// TIA Portal V16 export
// export: Created 2023-10-30T22:43:47.694868Z, ExportSetting WithDefaults, DisplayName Totally Integrated Automation Portal, DisplayVersion V16, DisplayName TIA Portal Version Control Interface, DisplayVersion V16, DisplayName TIA Portal Openness, DisplayVersion V16, DisplayName SINAMICS Startdrive Advanced, DisplayVersion V16, DisplayName SINAMICS Startdrive G130, G150, S120, S150, SINAMICS MV, S210, DisplayVersion V16, DisplayName SINAMICS Startdrive G110M, G120, G120C, G120D, G120P, DisplayVersion V16, DisplayName STEP 7 Professional, DisplayVersion V16, DisplayName STEP 7 Safety, DisplayVersion V16, DisplayName WinCC Professional, DisplayVersion V16
ORGANIZATION_BLOCK "Main"   // OB1, LAD, ProgramCycle
TITLE = "Main Program Sweep (Cycle)"
{ S7_Optimized_Access := 'TRUE' }
VERSION : 0.1
// stored: AutoNumber true, IsIECCheckEnabled false, SetENOAutomatically false
   VAR_INPUT
      Initial_Call : Bool;   // Initial call of this OB
      Remanence : Bool;   // =True, if remanent data are available
   END_VAR
   VAR_TEMP   // added for the SCL form of the ladder/FBD networks
      _w1 : Bool;
      _w2 : Bool;
      _w3 : Bool;
      _w4 : Bool;
   END_VAR
BEGIN

REGION Network 1: Control Maestro
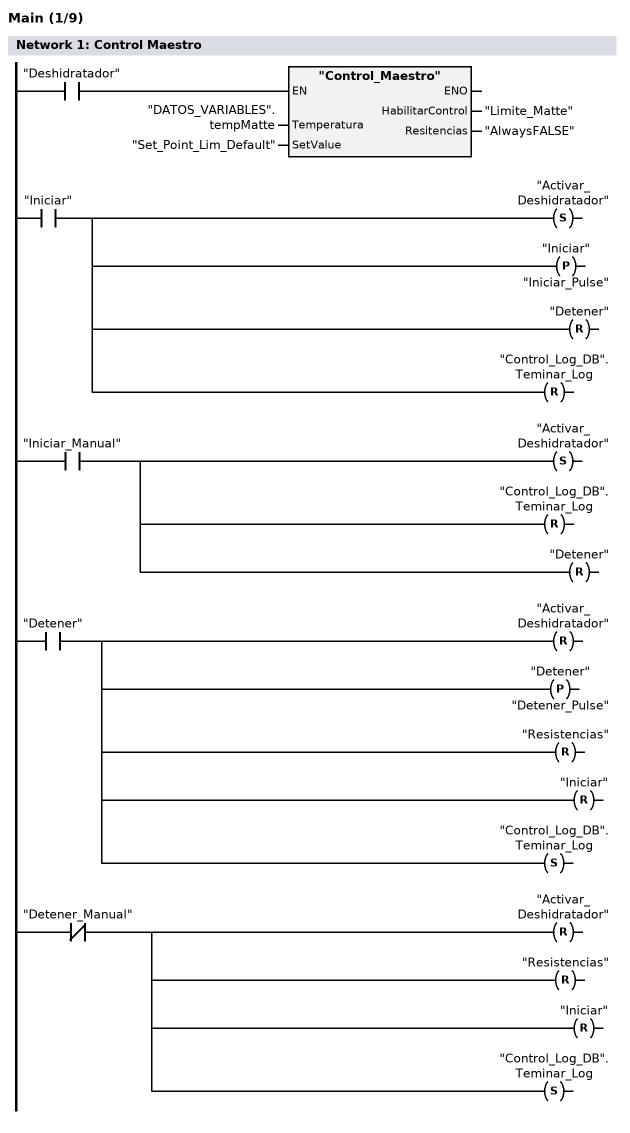
   IF "Deshidratador" THEN
       "Control_Maestro"(Temperatura := "DATOS_VARIABLES".tempMatte,
                         SetValue := "Set_Point_Lim_Default",
                         HabilitarControl => "Limite_Matte",
                         Resitencias => "AlwaysFALSE");
   END_IF;
   IF "Iniciar" THEN "Activar_Deshidratador" := TRUE; END_IF;
   #_w1 := "Iniciar";
   #_w2 := "Iniciar";
   "Iniciar" := #_w1 AND NOT "Iniciar_Pulse";   // rising edge
   "Iniciar_Pulse" := #_w1;
   IF #_w2 THEN
       "Detener" := FALSE;
       "Control_Log_DB".Teminar_Log := FALSE;
   END_IF;
   IF "Iniciar_Manual" THEN
       "Activar_Deshidratador" := TRUE;
       "Control_Log_DB".Teminar_Log := FALSE;
       "Detener" := FALSE;
   END_IF;
   IF "Detener" THEN "Activar_Deshidratador" := FALSE; END_IF;
   #_w3 := "Detener";
   #_w4 := "Detener";
   "Detener" := #_w3 AND NOT "Detener_Pulse";   // rising edge
   "Detener_Pulse" := #_w3;
   IF #_w4 THEN
       "Resistencias" := FALSE;
       "Iniciar" := FALSE;
       "Control_Log_DB".Teminar_Log := TRUE;
   END_IF;
   IF NOT "Detener_Manual" THEN
       "Activar_Deshidratador" := FALSE;
       "Resistencias" := FALSE;
       "Iniciar" := FALSE;
       "Control_Log_DB".Teminar_Log := TRUE;
   END_IF;
END_REGION

REGION Network 2: Matte
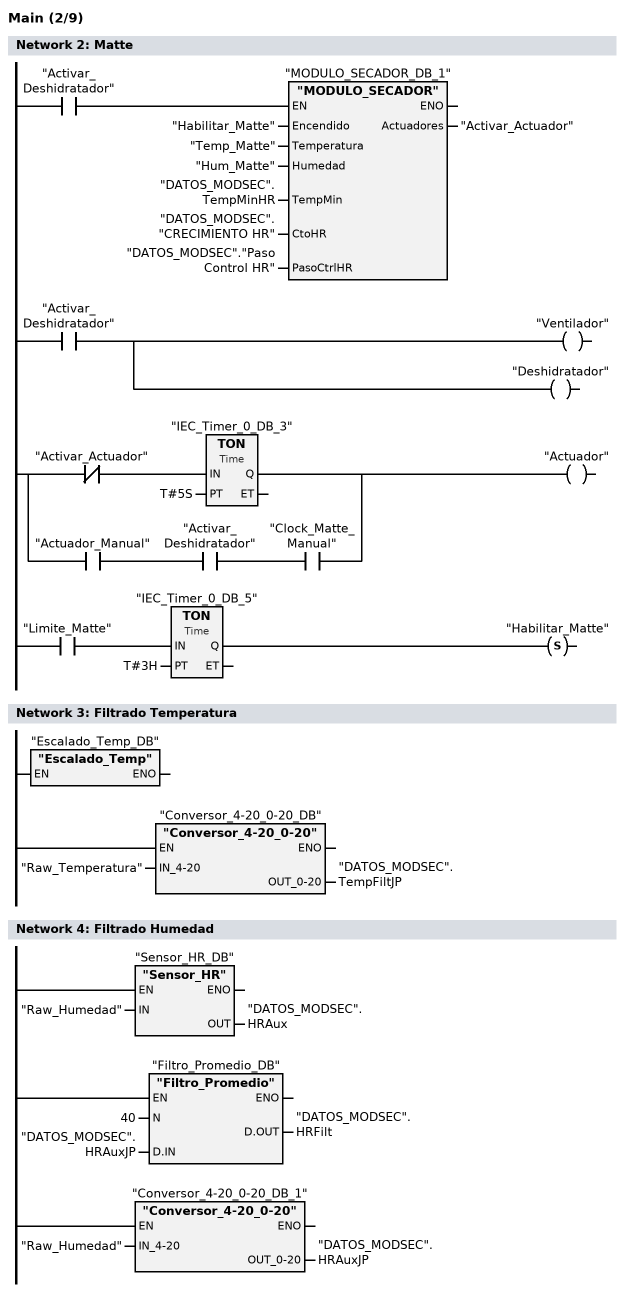
   RUNG wire#powerrail
      Contact( "Activar_Deshidratador" )
      "MODULO_SECADOR_DB_1"(Encendido := "Habilitar_Matte", Temperatura := "Temp_Matte", Humedad := "Hum_Matte", TempMin := "DATOS_MODSEC".TempMinHR, CtoHR := "DATOS_MODSEC"."CRECIMIENTO HR", PasoCtrlHR := "DATOS_MODSEC"."Paso Control HR", Actuadores => "Activar_Actuador")
   END_RUNG
   RUNG wire#powerrail
      Contact( "Activar_Deshidratador" )
      wire#w1
      Coil( "Ventilador" )
   END_RUNG
   RUNG wire#w1
      Coil( "Deshidratador" )
   END_RUNG
   RUNG wire#powerrail
      I_Contact( "Activar_Actuador" )
      { S7_Templates := "time_type := Time" } "IEC_Timer_0_DB_3".TON(pt := T#5S, et =>)
      wire#w2
      Coil( "Actuador" )
   END_RUNG
   RUNG wire#powerrail
      Contact( "Actuador_Manual" )
      Contact( "Activar_Deshidratador" )
      Contact( "Clock_Matte_Manual" )
   END_RUNG wire#w2
   RUNG wire#powerrail
      Contact( "Limite_Matte" )
      { S7_Templates := "time_type := Time" } "IEC_Timer_0_DB_5".TON(pt := T#3H, et =>)
      S_Coil( "Habilitar_Matte" )
   END_RUNG
   // the same network as SCL:
   IF "Activar_Deshidratador" THEN
       "MODULO_SECADOR_DB_1"(Encendido := "Habilitar_Matte",   // "MODULO_SECADOR"
                             Temperatura := "Temp_Matte",
                             Humedad := "Hum_Matte",
                             TempMin := "DATOS_MODSEC".TempMinHR,
                             CtoHR := "DATOS_MODSEC"."CRECIMIENTO HR",
                             PasoCtrlHR := "DATOS_MODSEC"."Paso Control HR",
                             Actuadores => "Activar_Actuador");
   END_IF;
   "Ventilador" := "Activar_Deshidratador";
   "Deshidratador" := "Activar_Deshidratador";
   "IEC_Timer_0_DB_3".TON(IN := NOT "Activar_Actuador", PT := T#5S);
   "Actuador" := "IEC_Timer_0_DB_3".Q OR ("Actuador_Manual" AND "Activar_Deshidratador" AND "Clock_Matte_Manual");
   "IEC_Timer_0_DB_5".TON(IN := "Limite_Matte", PT := T#3H);
   IF "IEC_Timer_0_DB_5".Q THEN "Habilitar_Matte" := TRUE; END_IF;
END_REGION

REGION Network 3: Filtrado Temperatura
   RUNG wire#powerrail
      "Escalado_Temp_DB"()
   END_RUNG
   RUNG wire#powerrail
      "Conversor_4-20_0-20_DB"("IN_4-20" := "Raw_Temperatura", "OUT_0-20" => "DATOS_MODSEC".TempFiltJP)
   END_RUNG
   // the same network as SCL:
   "Escalado_Temp_DB"();   // "Escalado_Temp"
   "Conversor_4-20_0-20_DB"("IN_4-20" := "Raw_Temperatura", "OUT_0-20" => "DATOS_MODSEC".TempFiltJP);   // "Conversor_4-20_0-20"
END_REGION

REGION Network 4: Filtrado Humedad
   RUNG wire#powerrail
      "Sensor_HR_DB"(IN := "Raw_Humedad", OUT => "DATOS_MODSEC".HRAux)
   END_RUNG
   RUNG wire#powerrail
      "Filtro_Promedio_DB"(N := 40, "D.IN" := "DATOS_MODSEC".HRAuxJP, "D.OUT" => "DATOS_MODSEC".HRFilt)
   END_RUNG
   RUNG wire#powerrail
      "Conversor_4-20_0-20_DB_1"("IN_4-20" := "Raw_Humedad", "OUT_0-20" => "DATOS_MODSEC".HRAuxJP)
   END_RUNG
   // the same network as SCL:
   "Sensor_HR_DB"(IN := "Raw_Humedad", OUT => "DATOS_MODSEC".HRAux);   // "Sensor_HR"
   "Filtro_Promedio_DB"(N := 40, "D.IN" := "DATOS_MODSEC".HRAuxJP, "D.OUT" => "DATOS_MODSEC".HRFilt);   // "Filtro_Promedio"
   "Conversor_4-20_0-20_DB_1"("IN_4-20" := "Raw_Humedad", "OUT_0-20" => "DATOS_MODSEC".HRAuxJP);   // "Conversor_4-20_0-20"
END_REGION

REGION Network 5: Simulación
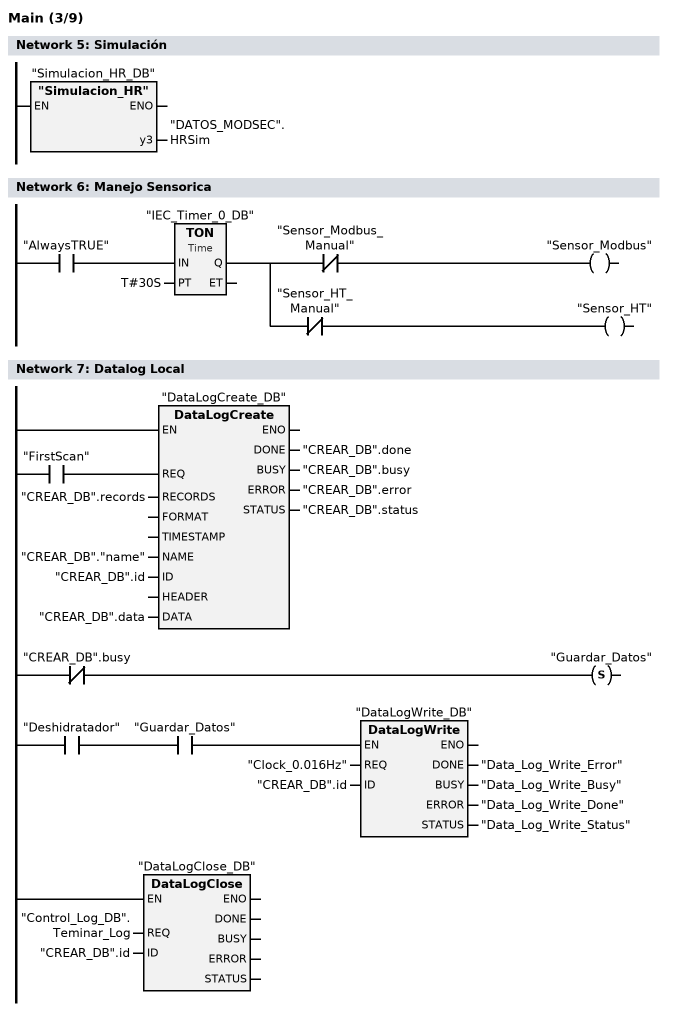
   RUNG wire#powerrail
      "Simulacion_HR_DB"(y3 => "DATOS_MODSEC".HRSim)
   END_RUNG
   // the same network as SCL:
   "Simulacion_HR_DB"(y3 => "DATOS_MODSEC".HRSim);   // "Simulacion_HR"
END_REGION

REGION Network 6: Manejo Sensorica
   RUNG wire#powerrail
      Contact( "AlwaysTRUE" )
      { S7_Templates := "time_type := Time" } "IEC_Timer_0_DB".TON(pt := T#30S, et =>)
      wire#w1
      I_Contact( "Sensor_Modbus_Manual" )
      Coil( "Sensor_Modbus" )
   END_RUNG
   RUNG wire#w1
      I_Contact( "Sensor_HT_Manual" )
      Coil( "Sensor_HT" )
   END_RUNG
   // the same network as SCL:
   "IEC_Timer_0_DB".TON(IN := "AlwaysTRUE", PT := T#30S);
   "Sensor_Modbus" := "IEC_Timer_0_DB".Q AND NOT "Sensor_Modbus_Manual";
   "Sensor_HT" := "IEC_Timer_0_DB".Q AND NOT "Sensor_HT_Manual";
END_REGION

REGION Network 7: Datalog Local
   RUNG wire#powerrail
      "DataLogCreate_DB".DataLogCreate(REQ := wire#w1, RECORDS := "CREAR_DB".records, FORMAT :=, TIMESTAMP :=, "NAME" := "CREAR_DB"."name", ID := "CREAR_DB".id, HEADER :=, DATA := "CREAR_DB".data, DONE => "CREAR_DB".done, BUSY => "CREAR_DB".busy, ERROR => "CREAR_DB".error, STATUS => "CREAR_DB".status)
   END_RUNG
   RUNG wire#powerrail
      Contact( "FirstScan" )
   END_RUNG wire#w1
   RUNG wire#powerrail
      I_Contact( "CREAR_DB".busy )
      S_Coil( "Guardar_Datos" )
   END_RUNG
   RUNG wire#powerrail
      Contact( "Deshidratador" )
      Contact( "Guardar_Datos" )
      "DataLogWrite_DB".DataLogWrite(REQ := "Clock_0.016Hz", ID := "CREAR_DB".id, DONE => "Data_Log_Write_Error", BUSY => "Data_Log_Write_Busy", ERROR => "Data_Log_Write_Done", STATUS => "Data_Log_Write_Status")
   END_RUNG
   RUNG wire#powerrail
      "DataLogClose_DB".DataLogClose(REQ := "Control_Log_DB".Teminar_Log, ID := "CREAR_DB".id, DONE =>, BUSY =>, ERROR =>, STATUS =>)
   END_RUNG
   // the same network as SCL:
   "DataLogCreate_DB"(REQ := "FirstScan",   // DataLogCreate
                      RECORDS := "CREAR_DB".records,
                      "NAME" := "CREAR_DB"."name",
                      ID := "CREAR_DB".id,
                      DATA := "CREAR_DB".data,
                      DONE => "CREAR_DB".done,
                      BUSY => "CREAR_DB".busy,
                      ERROR => "CREAR_DB".error,
                      STATUS => "CREAR_DB".status);
   IF NOT "CREAR_DB".busy THEN "Guardar_Datos" := TRUE; END_IF;
   IF "Deshidratador" AND "Guardar_Datos" THEN
       "DataLogWrite_DB"(REQ := "Clock_0.016Hz",   // DataLogWrite
                         ID := "CREAR_DB".id,
                         DONE => "Data_Log_Write_Error",
                         BUSY => "Data_Log_Write_Busy",
                         ERROR => "Data_Log_Write_Done",
                         STATUS => "Data_Log_Write_Status");
   END_IF;
   "DataLogClose_DB"(REQ := "Control_Log_DB".Teminar_Log, ID := "CREAR_DB".id);   // DataLogClose
END_REGION

REGION Network 8: Mover Datos para Log Remoto
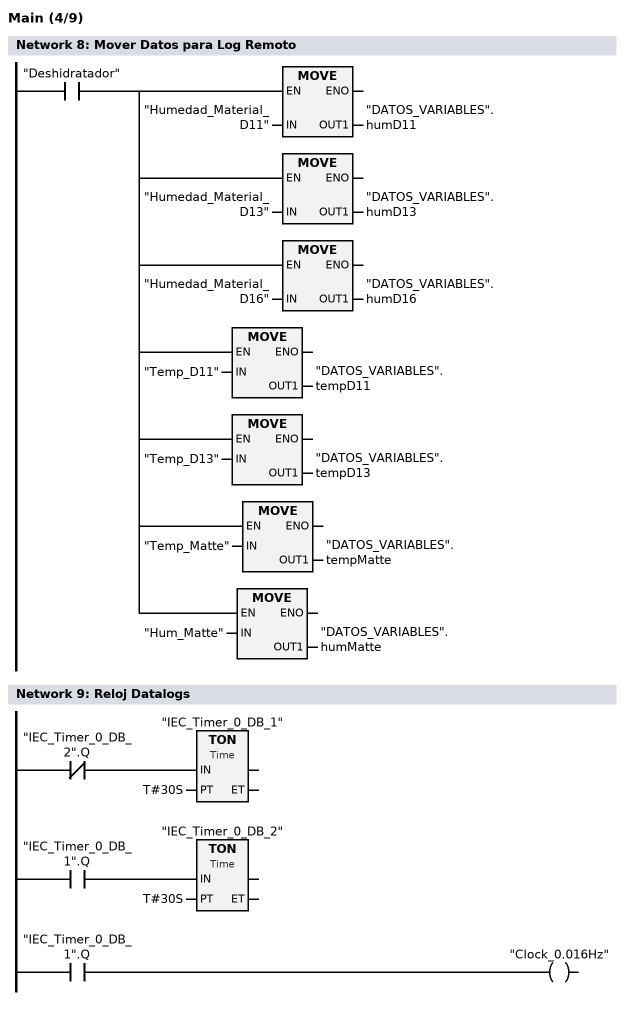
   RUNG wire#powerrail
      Contact( "Deshidratador" )
      wire#w1
      Move(in := "Humedad_Material_D11", out1 => "DATOS_VARIABLES".humD11)
   END_RUNG
   RUNG wire#w1
      Move(in := "Humedad_Material_D13", out1 => "DATOS_VARIABLES".humD13)
   END_RUNG
   RUNG wire#w1
      Move(in := "Humedad_Material_D16", out1 => "DATOS_VARIABLES".humD16)
   END_RUNG
   RUNG wire#w1
      Move(in := "Temp_D11", out1 => "DATOS_VARIABLES".tempD11)
   END_RUNG
   RUNG wire#w1
      Move(in := "Temp_D13", out1 => "DATOS_VARIABLES".tempD13)
   END_RUNG
   RUNG wire#w1
      Move(in := "Temp_Matte", out1 => "DATOS_VARIABLES".tempMatte)
   END_RUNG
   RUNG wire#w1
      Move(in := "Hum_Matte", out1 => "DATOS_VARIABLES".humMatte)
   END_RUNG
   // the same network as SCL:
   IF "Deshidratador" THEN
       "DATOS_VARIABLES".humD11 := "Humedad_Material_D11";
       "DATOS_VARIABLES".humD13 := "Humedad_Material_D13";
       "DATOS_VARIABLES".humD16 := "Humedad_Material_D16";
       "DATOS_VARIABLES".tempD11 := "Temp_D11";
       "DATOS_VARIABLES".tempD13 := "Temp_D13";
       "DATOS_VARIABLES".tempMatte := "Temp_Matte";
       "DATOS_VARIABLES".humMatte := "Hum_Matte";
   END_IF;
END_REGION

REGION Network 9: Reloj Datalogs
   RUNG wire#powerrail
      I_Contact( "IEC_Timer_0_DB_2".Q )
      { S7_Templates := "time_type := Time" } "IEC_Timer_0_DB_1".TON(pt := T#30S, et =>)
   END_RUNG
   RUNG wire#powerrail
      Contact( "IEC_Timer_0_DB_1".Q )
      { S7_Templates := "time_type := Time" } "IEC_Timer_0_DB_2".TON(pt := T#30S, et =>)
   END_RUNG
   RUNG wire#powerrail
      Contact( "IEC_Timer_0_DB_1".Q )
      Coil( "Clock_0.016Hz" )
   END_RUNG
   // the same network as SCL:
   "IEC_Timer_0_DB_1".TON(IN := NOT "IEC_Timer_0_DB_2".Q, PT := T#30S);
   "IEC_Timer_0_DB_2".TON(IN := "IEC_Timer_0_DB_1".Q, PT := T#30S);
   "Clock_0.016Hz" := "IEC_Timer_0_DB_1".Q;
END_REGION

REGION Network 10: Mover Datos para Log Local
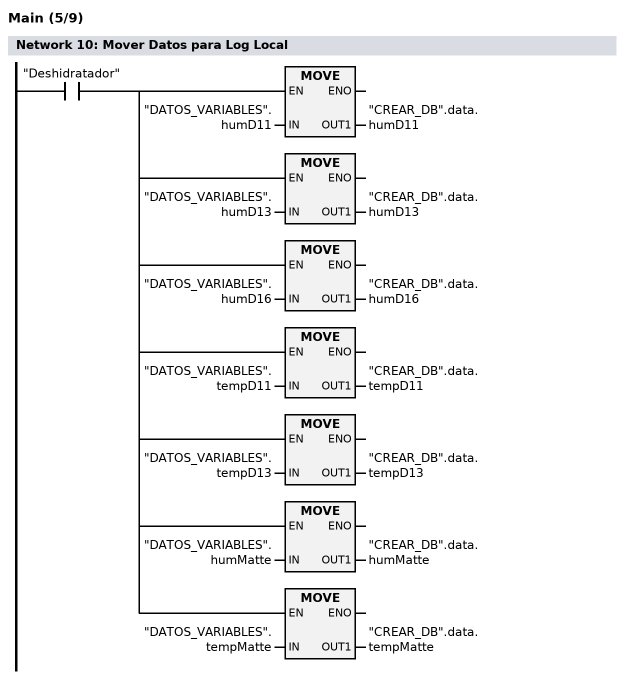
   RUNG wire#powerrail
      Contact( "Deshidratador" )
      wire#w1
      Move(in := "DATOS_VARIABLES".humD11, out1 => "CREAR_DB".data.humD11)
   END_RUNG
   RUNG wire#w1
      Move(in := "DATOS_VARIABLES".humD13, out1 => "CREAR_DB".data.humD13)
   END_RUNG
   RUNG wire#w1
      Move(in := "DATOS_VARIABLES".humD16, out1 => "CREAR_DB".data.humD16)
   END_RUNG
   RUNG wire#w1
      Move(in := "DATOS_VARIABLES".tempD11, out1 => "CREAR_DB".data.tempD11)
   END_RUNG
   RUNG wire#w1
      Move(in := "DATOS_VARIABLES".tempD13, out1 => "CREAR_DB".data.tempD13)
   END_RUNG
   RUNG wire#w1
      Move(in := "DATOS_VARIABLES".humMatte, out1 => "CREAR_DB".data.humMatte)
   END_RUNG
   RUNG wire#w1
      Move(in := "DATOS_VARIABLES".tempMatte, out1 => "CREAR_DB".data.tempMatte)
   END_RUNG
   // the same network as SCL:
   IF "Deshidratador" THEN
       "CREAR_DB".data.humD11 := "DATOS_VARIABLES".humD11;
       "CREAR_DB".data.humD13 := "DATOS_VARIABLES".humD13;
       "CREAR_DB".data.humD16 := "DATOS_VARIABLES".humD16;
       "CREAR_DB".data.tempD11 := "DATOS_VARIABLES".tempD11;
       "CREAR_DB".data.tempD13 := "DATOS_VARIABLES".tempD13;
       "CREAR_DB".data.humMatte := "DATOS_VARIABLES".humMatte;
       "CREAR_DB".data.tempMatte := "DATOS_VARIABLES".tempMatte;
   END_IF;
END_REGION

REGION Network 11: Comunicación Modbus
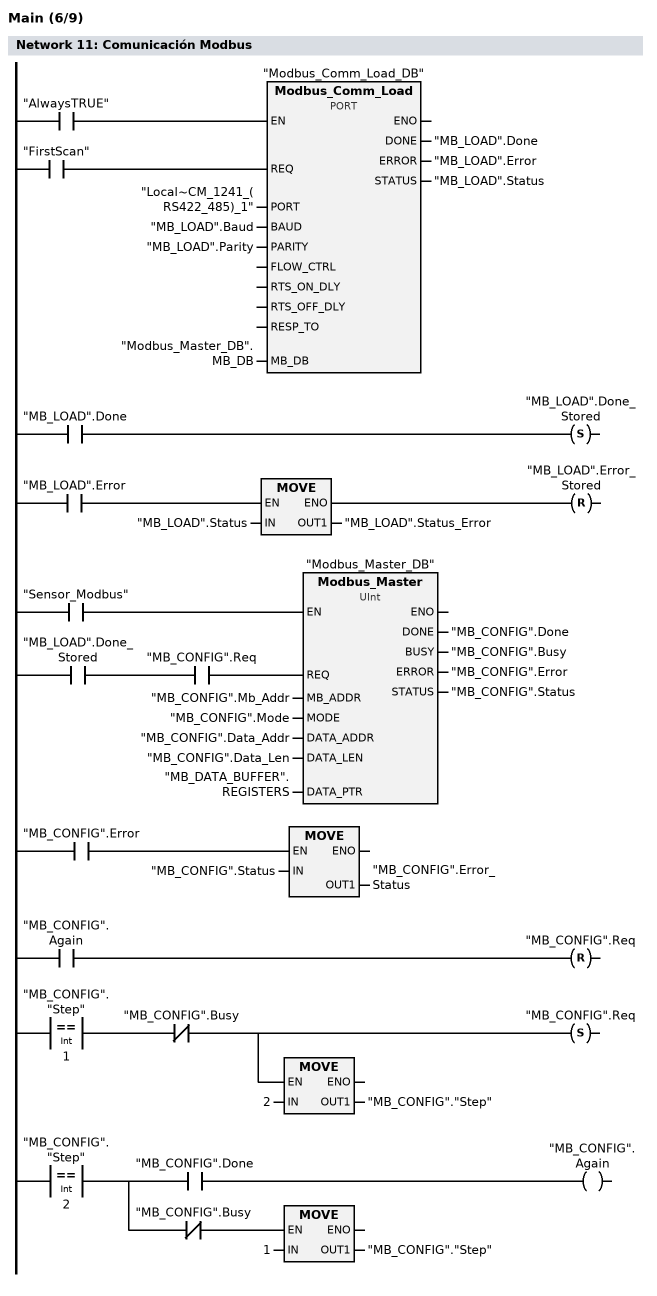
   RUNG wire#powerrail
      Contact( "AlwaysTRUE" )
      { S7_Templates := "[card := 0, port_type := PORT, word_type := UInt, dint_type := UDInt, mbbase_type := P2P_MB_BASE]" } "Modbus_Comm_Load_DB".Modbus_Comm_Load(REQ := wire#w1, PORT := "Local~CM_1241_(RS422_485)_1", BAUD := "MB_LOAD".Baud, PARITY := "MB_LOAD".Parity, FLOW_CTRL :=, RTS_ON_DLY :=, RTS_OFF_DLY :=, RESP_TO :=, MB_DB := "Modbus_Master_DB".MB_DB, DONE => "MB_LOAD".Done, ERROR => "MB_LOAD".Error, STATUS => "MB_LOAD".Status)
   END_RUNG
   RUNG wire#powerrail
      Contact( "FirstScan" )
   END_RUNG wire#w1
   RUNG wire#powerrail
      Contact( "MB_LOAD".Done )
      S_Coil( "MB_LOAD".Done_Stored )
   END_RUNG
   RUNG wire#powerrail
      Contact( "MB_LOAD".Error )
      Move(in := "MB_LOAD".Status, out1 => "MB_LOAD".Status_Error)
      R_Coil( "MB_LOAD".Error_Stored )
   END_RUNG
   RUNG wire#powerrail
      Contact( "Sensor_Modbus" )
      { S7_Templates := "[card := 0, word_type := UInt, dword_type := UDInt, byte_type := USInt, any_type := Variant]" } "Modbus_Master_DB".Modbus_Master(REQ := wire#w2, MB_ADDR := "MB_CONFIG".Mb_Addr, MODE := "MB_CONFIG".Mode, DATA_ADDR := "MB_CONFIG".Data_Addr, DATA_LEN := "MB_CONFIG".Data_Len, DATA_PTR := "MB_DATA_BUFFER".REGISTERS, DONE => "MB_CONFIG".Done, BUSY => "MB_CONFIG".Busy, ERROR => "MB_CONFIG".Error, STATUS => "MB_CONFIG".Status)
   END_RUNG
   RUNG wire#powerrail
      Contact( "MB_LOAD".Done_Stored )
      Contact( "MB_CONFIG".Req )
   END_RUNG wire#w2
   RUNG wire#powerrail
      Contact( "MB_CONFIG".Error )
      Move(in := "MB_CONFIG".Status, out1 => "MB_CONFIG".Error_Status)
   END_RUNG
   RUNG wire#powerrail
      Contact( "MB_CONFIG".Again )
      R_Coil( "MB_CONFIG".Req )
   END_RUNG
   RUNG wire#powerrail
      { S7_Templates := "SrcType := Int" } EQ_Contact(in1 := "MB_CONFIG"."Step", in2 := 1)
      I_Contact( "MB_CONFIG".Busy )
      wire#w3
      S_Coil( "MB_CONFIG".Req )
   END_RUNG
   RUNG wire#w3
      Move(in := 2, out1 => "MB_CONFIG"."Step")
   END_RUNG
   RUNG wire#powerrail
      { S7_Templates := "SrcType := Int" } EQ_Contact(in1 := "MB_CONFIG"."Step", in2 := 2)
      wire#w4
      Contact( "MB_CONFIG".Done )
      Coil( "MB_CONFIG".Again )
   END_RUNG
   RUNG wire#w4
      I_Contact( "MB_CONFIG".Busy )
      Move(in := 1, out1 => "MB_CONFIG"."Step")
   END_RUNG
   // the same network as SCL:
   IF "AlwaysTRUE" THEN
       "Modbus_Comm_Load_DB"(REQ := "FirstScan",   // Modbus_Comm_Load
                             PORT := "Local~CM_1241_(RS422_485)_1",
                             BAUD := "MB_LOAD".Baud,
                             PARITY := "MB_LOAD".Parity,
                             MB_DB := "Modbus_Master_DB".MB_DB,
                             DONE => "MB_LOAD".Done,
                             ERROR => "MB_LOAD".Error,
                             STATUS => "MB_LOAD".Status);
   END_IF;
   IF "MB_LOAD".Done THEN "MB_LOAD".Done_Stored := TRUE; END_IF;
   IF "MB_LOAD".Error THEN
       "MB_LOAD".Status_Error := "MB_LOAD".Status;
       "MB_LOAD".Error_Stored := FALSE;
   END_IF;
   IF "Sensor_Modbus" THEN
       "Modbus_Master_DB"(REQ := "MB_LOAD".Done_Stored AND "MB_CONFIG".Req,   // Modbus_Master
                          MB_ADDR := "MB_CONFIG".Mb_Addr,
                          MODE := "MB_CONFIG".Mode,
                          DATA_ADDR := "MB_CONFIG".Data_Addr,
                          DATA_LEN := "MB_CONFIG".Data_Len,
                          DATA_PTR := "MB_DATA_BUFFER".REGISTERS,
                          DONE => "MB_CONFIG".Done,
                          BUSY => "MB_CONFIG".Busy,
                          ERROR => "MB_CONFIG".Error,
                          STATUS => "MB_CONFIG".Status);
   END_IF;
   IF "MB_CONFIG".Error THEN "MB_CONFIG".Error_Status := "MB_CONFIG".Status; END_IF;
   IF "MB_CONFIG".Again THEN "MB_CONFIG".Req := FALSE; END_IF;
   IF ("MB_CONFIG"."Step" = 1) AND NOT "MB_CONFIG".Busy THEN
       "MB_CONFIG".Req := TRUE;
       "MB_CONFIG"."Step" := 2;
   END_IF;
   #_w1 := "MB_CONFIG"."Step" = 2;
   "MB_CONFIG".Again := #_w1 AND "MB_CONFIG".Done;
   IF #_w1 AND NOT "MB_CONFIG".Busy THEN "MB_CONFIG"."Step" := 1; END_IF;
END_REGION

REGION Network 12: Escalización Humedad
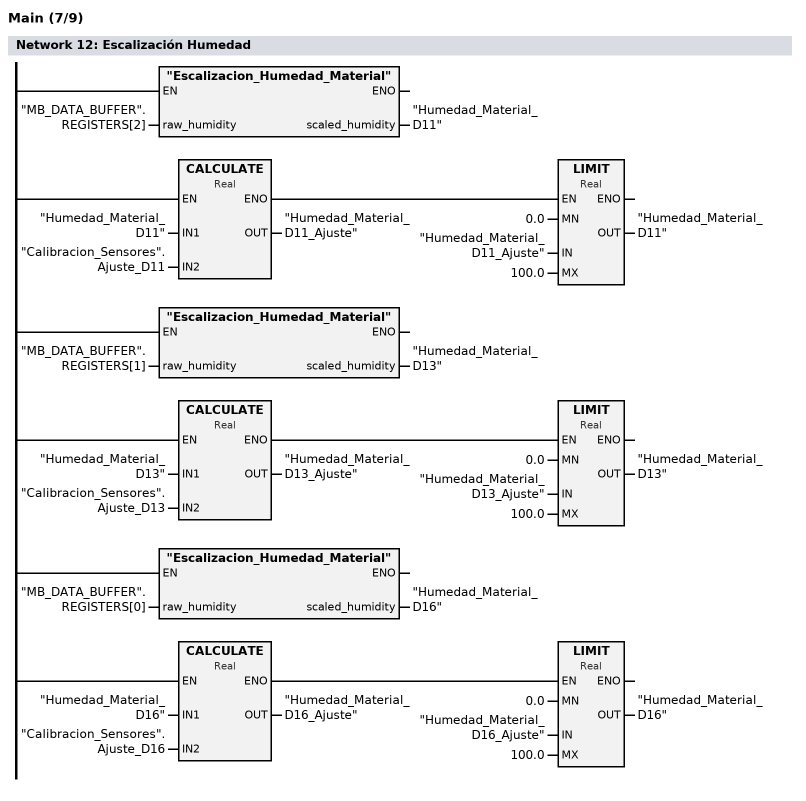
   RUNG wire#powerrail
      "Escalizacion_Humedad_Material"(raw_humidity := "MB_DATA_BUFFER".REGISTERS[2], scaled_humidity => "Humedad_Material_D11")
   END_RUNG
   RUNG wire#powerrail
      { S7_Templates := "SrcType := Real"; S7_Expression := "IN1 - IN2" } Calculate(in1 := "Humedad_Material_D11", in2 := "Calibracion_Sensores".Ajuste_D11, out => "Humedad_Material_D11_Ajuste")
      { S7_Templates := "value_type := Real" } Limit(mn := 0.0, in := "Humedad_Material_D11_Ajuste", mx := 100.0, out => "Humedad_Material_D11")
   END_RUNG
   RUNG wire#powerrail
      "Escalizacion_Humedad_Material"(raw_humidity := "MB_DATA_BUFFER".REGISTERS[1], scaled_humidity => "Humedad_Material_D13")
   END_RUNG
   RUNG wire#powerrail
      { S7_Templates := "SrcType := Real"; S7_Expression := "IN1 - IN2" } Calculate(in1 := "Humedad_Material_D13", in2 := "Calibracion_Sensores".Ajuste_D13, out => "Humedad_Material_D13_Ajuste")
      { S7_Templates := "value_type := Real" } Limit(mn := 0.0, in := "Humedad_Material_D13_Ajuste", mx := 100.0, out => "Humedad_Material_D13")
   END_RUNG
   RUNG wire#powerrail
      "Escalizacion_Humedad_Material"(raw_humidity := "MB_DATA_BUFFER".REGISTERS[0], scaled_humidity => "Humedad_Material_D16")
   END_RUNG
   RUNG wire#powerrail
      { S7_Templates := "SrcType := Real"; S7_Expression := "IN1 - IN2" } Calculate(in1 := "Humedad_Material_D16", in2 := "Calibracion_Sensores".Ajuste_D16, out => "Humedad_Material_D16_Ajuste")
      { S7_Templates := "value_type := Real" } Limit(mn := 0.0, in := "Humedad_Material_D16_Ajuste", mx := 100.0, out => "Humedad_Material_D16")
   END_RUNG
   // the same network as SCL:
   "Escalizacion_Humedad_Material"(raw_humidity := "MB_DATA_BUFFER".REGISTERS[2],
                           scaled_humidity => "Humedad_Material_D11");
   "Humedad_Material_D11_Ajuste" := "Humedad_Material_D11" - "Calibracion_Sensores".Ajuste_D11;
   "Humedad_Material_D11" := LIMIT(MN := 0.0, IN := "Humedad_Material_D11_Ajuste", MX := 100.0);
   "Escalizacion_Humedad_Material"(raw_humidity := "MB_DATA_BUFFER".REGISTERS[1],
                           scaled_humidity => "Humedad_Material_D13");
   "Humedad_Material_D13_Ajuste" := "Humedad_Material_D13" - "Calibracion_Sensores".Ajuste_D13;
   "Humedad_Material_D13" := LIMIT(MN := 0.0, IN := "Humedad_Material_D13_Ajuste", MX := 100.0);
   "Escalizacion_Humedad_Material"(raw_humidity := "MB_DATA_BUFFER".REGISTERS[0],
                           scaled_humidity => "Humedad_Material_D16");
   "Humedad_Material_D16_Ajuste" := "Humedad_Material_D16" - "Calibracion_Sensores".Ajuste_D16;
   "Humedad_Material_D16" := LIMIT(MN := 0.0, IN := "Humedad_Material_D16_Ajuste", MX := 100.0);
END_REGION

REGION Network 13: Humedad y Temperatura Deshidratador
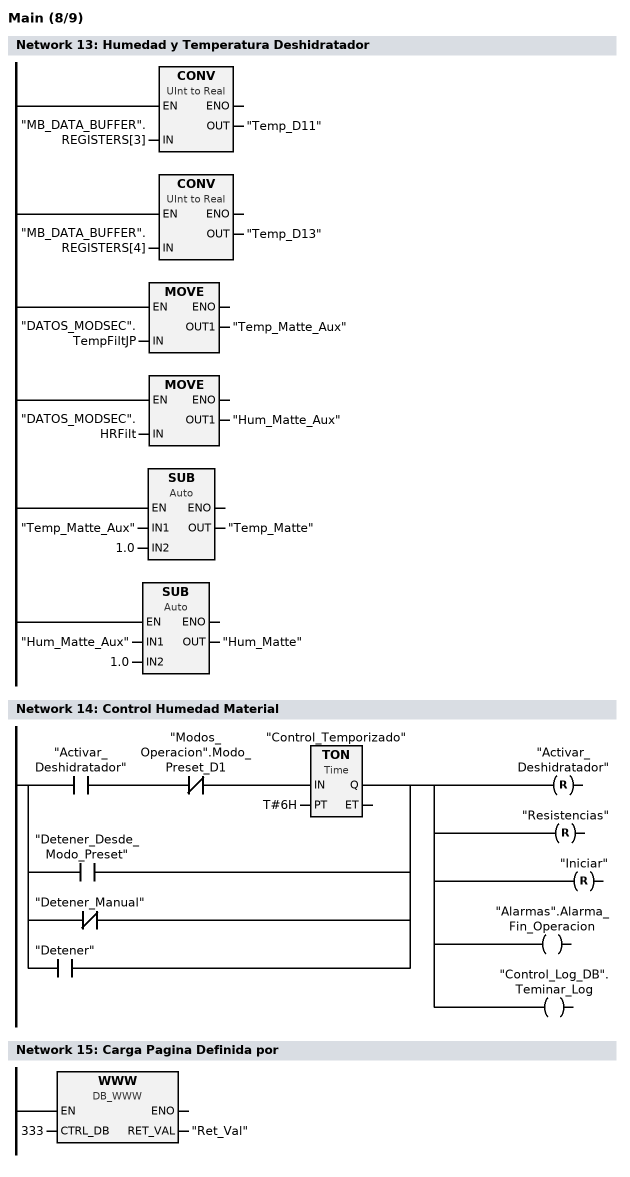
   RUNG wire#powerrail
      { S7_Templates := "[SrcType := UInt, DestType := Real]" } Convert(in := "MB_DATA_BUFFER".REGISTERS[3], out => "Temp_D11")
   END_RUNG
   RUNG wire#powerrail
      { S7_Templates := "[SrcType := UInt, DestType := Real]" } Convert(in := "MB_DATA_BUFFER".REGISTERS[4], out => "Temp_D13")
   END_RUNG
   RUNG wire#powerrail
      Move(in := "DATOS_MODSEC".TempFiltJP, out1 => "Temp_Matte_Aux")
   END_RUNG
   RUNG wire#powerrail
      Move(in := "DATOS_MODSEC".HRFilt, out1 => "Hum_Matte_Aux")
   END_RUNG
   RUNG wire#powerrail
      Sub(in1 := "Temp_Matte_Aux", in2 := 1.0, out => "Temp_Matte")
   END_RUNG
   RUNG wire#powerrail
      Sub(in1 := "Hum_Matte_Aux", in2 := 1.0, out => "Hum_Matte")
   END_RUNG
   // the same network as SCL:
   "Temp_D11" := UINT_TO_REAL("MB_DATA_BUFFER".REGISTERS[3]);
   "Temp_D13" := UINT_TO_REAL("MB_DATA_BUFFER".REGISTERS[4]);
   "Temp_Matte_Aux" := "DATOS_MODSEC".TempFiltJP;
   "Hum_Matte_Aux" := "DATOS_MODSEC".HRFilt;
   "Temp_Matte" := "Temp_Matte_Aux" - 1.0;
   "Hum_Matte" := "Hum_Matte_Aux" - 1.0;
END_REGION

REGION Network 14: Control Humedad Material
   RUNG wire#powerrail
      Contact( "Activar_Deshidratador" )
      I_Contact( "Modos_Operacion".Modo_Preset_D1 )
      { S7_Templates := "time_type := Time" } "Control_Temporizado".TON(pt := T#6H, et =>)
      wire#w1
      R_Coil( "Activar_Deshidratador" )
   END_RUNG
   RUNG wire#powerrail
      Contact( "Detener_Desde_Modo_Preset" )
   END_RUNG wire#w1
   RUNG wire#powerrail
      I_Contact( "Detener_Manual" )
   END_RUNG wire#w1
   RUNG wire#powerrail
      Contact( "Detener" )
   END_RUNG wire#w1
   RUNG wire#w1
      R_Coil( "Resistencias" )
   END_RUNG
   RUNG wire#w1
      R_Coil( "Iniciar" )
   END_RUNG
   RUNG wire#w1
      Coil( "Alarmas".Alarma_Fin_Operacion )
   END_RUNG
   RUNG wire#w1
      Coil( "Control_Log_DB".Teminar_Log )
   END_RUNG
   // the same network as SCL:
   "Control_Temporizado".TON(IN := "Activar_Deshidratador" AND NOT "Modos_Operacion".Modo_Preset_D1, PT := T#6H);
   #_w1 := "Control_Temporizado".Q OR "Detener_Desde_Modo_Preset" OR NOT "Detener_Manual" OR "Detener";
   IF #_w1 THEN
       "Activar_Deshidratador" := FALSE;
       "Resistencias" := FALSE;
       "Iniciar" := FALSE;
   END_IF;
   "Alarmas".Alarma_Fin_Operacion := #_w1;
   "Control_Log_DB".Teminar_Log := #_w1;
END_REGION

REGION Network 15: Carga Pagina Definida por
   RUNG wire#powerrail
      { S7_Templates := "value_type := DB_WWW" } WWW(CTRL_DB := 333, RET_VAL => "Ret_Val")
   END_RUNG
   // the same network as SCL:
   "Ret_Val" := WWW(CTRL_DB := 333);
END_REGION

REGION Network 16: Matte Modo Manual
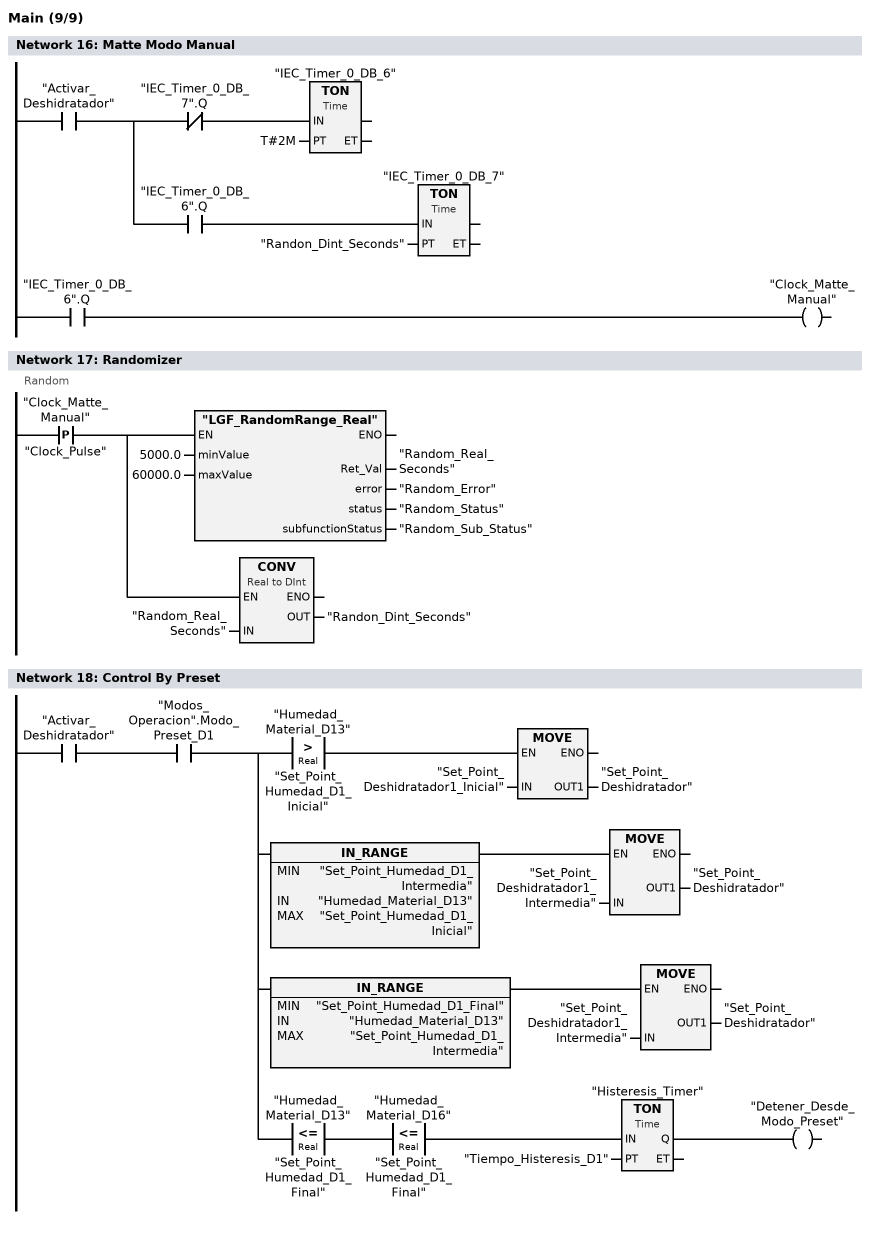
   RUNG wire#powerrail
      Contact( "Activar_Deshidratador" )
      wire#w1
      I_Contact( "IEC_Timer_0_DB_7".Q )
      { S7_Templates := "time_type := Time" } "IEC_Timer_0_DB_6".TON(pt := T#2M, et =>)
   END_RUNG
   RUNG wire#w1
      Contact( "IEC_Timer_0_DB_6".Q )
      { S7_Templates := "time_type := Time" } "IEC_Timer_0_DB_7".TON(pt := "Randon_Dint_Seconds", et =>)
   END_RUNG
   RUNG wire#powerrail
      Contact( "IEC_Timer_0_DB_6".Q )
      Coil( "Clock_Matte_Manual" )
   END_RUNG
   // the same network as SCL:
   "IEC_Timer_0_DB_6".TON(IN := "Activar_Deshidratador" AND NOT "IEC_Timer_0_DB_7".Q, PT := T#2M);
   "IEC_Timer_0_DB_7".TON(IN := "Activar_Deshidratador" AND "IEC_Timer_0_DB_6".Q, PT := "Randon_Dint_Seconds");
   "Clock_Matte_Manual" := "IEC_Timer_0_DB_6".Q;
END_REGION

REGION Network 17: Randomizer
   // Random
   RUNG wire#powerrail
      P_Contact(operand := "Clock_Matte_Manual", bit := "Clock_Pulse")
      wire#w1
      "LGF_RandomRange_Real"(minValue := 5000.0, maxValue := 60000.0, Ret_Val => "Random_Real_Seconds", error => "Random_Error", status => "Random_Status", subfunctionStatus => "Random_Sub_Status")
   END_RUNG
   RUNG wire#w1
      { S7_Templates := "[SrcType := Real, DestType := DInt]" } Convert(in := "Random_Real_Seconds", out => "Randon_Dint_Seconds")
   END_RUNG
   // the same network as SCL:
   #_w1 := "Clock_Matte_Manual" AND NOT "Clock_Pulse";   // rising edge of "Clock_Matte_Manual"
   "Clock_Pulse" := "Clock_Matte_Manual";
   IF #_w1 THEN
       "Random_Real_Seconds" := "LGF_RandomRange_Real"(minValue := 5000.0,
                               maxValue := 60000.0,
                               error => "Random_Error",
                               status => "Random_Status",
                               subfunctionStatus => "Random_Sub_Status");
       "Randon_Dint_Seconds" := REAL_TO_DINT("Random_Real_Seconds");
   END_IF;
END_REGION

REGION Network 18: Control By Preset
   RUNG wire#powerrail
      Contact( "Activar_Deshidratador" )
      Contact( "Modos_Operacion".Modo_Preset_D1 )
      wire#w1
      { S7_Templates := "SrcType := Real" } GT_Contact(in1 := "Humedad_Material_D13", in2 := "Set_Point_Humedad_D1_Inicial")
      Move(in := "Set_Point_Deshidratador1_Inicial", out1 => "Set_Point_Deshidratador")
   END_RUNG
   RUNG wire#w1
      { S7_Templates := "SrcType := Real" } InRange(min := "Set_Point_Humedad_D1_Intermedia", in := "Humedad_Material_D13", max := "Set_Point_Humedad_D1_Inicial")
      Move(in := "Set_Point_Deshidratador1_Intermedia", out1 => "Set_Point_Deshidratador")
   END_RUNG
   RUNG wire#w1
      { S7_Templates := "SrcType := Real" } InRange(min := "Set_Point_Humedad_D1_Final", in := "Humedad_Material_D13", max := "Set_Point_Humedad_D1_Intermedia")
      Move(in := "Set_Point_Deshidratador1_Intermedia", out1 => "Set_Point_Deshidratador")
   END_RUNG
   RUNG wire#w1
      { S7_Templates := "SrcType := Real" } LE_Contact(in1 := "Humedad_Material_D13", in2 := "Set_Point_Humedad_D1_Final")
      { S7_Templates := "SrcType := Real" } LE_Contact(in1 := "Humedad_Material_D16", in2 := "Set_Point_Humedad_D1_Final")
      { S7_Templates := "time_type := Time" } "Histeresis_Timer".TON(pt := "Tiempo_Histeresis_D1", et =>)
      Coil( "Detener_Desde_Modo_Preset" )
   END_RUNG
   // the same network as SCL:
   #_w1 := "Activar_Deshidratador" AND "Modos_Operacion".Modo_Preset_D1;
   IF #_w1 AND ("Humedad_Material_D13" > "Set_Point_Humedad_D1_Inicial") THEN
       "Set_Point_Deshidratador" := "Set_Point_Deshidratador1_Inicial";
   END_IF;
   IF #_w1 AND ("Set_Point_Humedad_D1_Intermedia" <= "Humedad_Material_D13") AND ("Humedad_Material_D13" <= "Set_Point_Humedad_D1_Inicial") THEN
       "Set_Point_Deshidratador" := "Set_Point_Deshidratador1_Intermedia";
   END_IF;
   IF #_w1 AND ("Set_Point_Humedad_D1_Final" <= "Humedad_Material_D13") AND ("Humedad_Material_D13" <= "Set_Point_Humedad_D1_Intermedia") THEN
       "Set_Point_Deshidratador" := "Set_Point_Deshidratador1_Intermedia";
   END_IF;
   "Histeresis_Timer".TON(IN := #_w1 AND ("Humedad_Material_D13" <= "Set_Point_Humedad_D1_Final") AND ("Humedad_Material_D16" <= "Set_Point_Humedad_D1_Final"),
                          PT := "Tiempo_Histeresis_D1");
   "Detener_Desde_Modo_Preset" := "Histeresis_Timer".Q;
END_REGION
END_ORGANIZATION_BLOCK
